//-----------------------------------------------------------------------------------------------------
//																
//									 	Tkmatik sp z o.o.
//
//	Name					:		FB_Load
//	Author					:		AM
//	Release Date			:		12.01.2022
//	Current ver				:		v 0.1
// 	Last correction 		:		12.01.2022
// 
//	Description				:
//		Special FB for loading structures from BINARY files						
//
//	Requared hardware		:
//
// 	Configuration			:
//
//
//-----------------------------------------------------------------------------------------------------

FUNCTION_BLOCK FB_Load
VAR_INPUT
	sFilePath											:	STRING(255);					//	File path (e.g. 'C:\1.txt')
	pStructAdr											:	PVOID;                          //	Pointer on data struct
	udiStructSize										:	UDINT;                          //	Size of datastruct
	bExecute											:	BOOL;                           //
END_VAR                                                                                     
VAR_OUTPUT                                                                                  
	bBusy												:	BOOL;                           //	FB is Busy
	bDone												:	BOOL;                           //	Load cycle done, DATA actual 
	bError												:	BOOL;                           //	Flag error
	nErrId												:	UDINT;                          //	Error ID
END_VAR                                                                                     
VAR                                                                                         
	fbFileOpen											:	FB_FileOpen;                    //	FB for opening 
	fbFileClose											:	FB_FileClose;                   //	FB for closing
	fbFileRead											:	FB_FileRead;                    //	FB for reading
	hFile												:	UINT;                           //	File hendler
	eMainCase											:	E_FileOpSteps;                  //	Main cycle case value
	rtExecute											:	R_TRIG;                         //	Rtrig for start
END_VAR

ACT_FBs();
ACT_Main();

ACTION ACT_FBs:
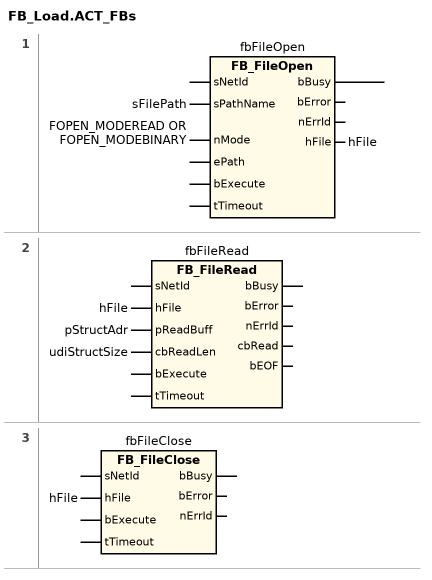
// NETWORK 1
fbFileOpen(sPathName := sFilePath, nMode := FOPEN_MODEREAD OR FOPEN_MODEBINARY, hFile => hFile); // FB_FileOpen

// NETWORK 2
fbFileRead(hFile := hFile, pReadBuff := pStructAdr, cbReadLen := udiStructSize); // FB_FileRead

// NETWORK 3
fbFileClose(hFile := hFile); // FB_FileClose
END_ACTION

ACTION ACT_Main:
rtExecute(CLK:=bExecute);
IF (NOT bExecute) THEN
	bDone												:=	FALSE;
END_IF

CASE eMainCase OF
	E_FileOpSteps.eNop:
		fbFileClose.bExecute							:=	FALSE;
		fbFileOpen.bExecute								:=	FALSE;
		fbFileRead.bExecute								:=	FALSE;
		bBusy											:=	FALSE;
		
		IF (rtExecute.Q) THEN
			bError										:=	FALSE;
			nErrId										:=	0;
			eMainCase									:=	E_FileOpSteps.eStartOpen;
			bBusy										:=	TRUE;
		END_IF
		
	E_FileOpSteps.eStartOpen:
		fbFileOpen.bExecute								:=	TRUE;
		eMainCase										:=	E_FileOpSteps.eWaitOpen;

	E_FileOpSteps.eWaitOpen:
		IF (fbFileOpen.bError) THEN
			bError										:=	TRUE;
			nErrId										:=	10;
			eMainCase									:=	E_FileOpSteps.eNop;
		ELSIF (NOT fbFileOpen.bBusy) THEN
			fbFileOpen.bExecute							:=	FALSE;
			eMainCase									:=	E_FileOpSteps.eStartOper;
		END_IF
		
	E_FileOpSteps.eStartOper:
		fbFileRead.bExecute								:=	TRUE;
		eMainCase										:=	E_FileOpSteps.eWaitOper;
		
	E_FileOpSteps.eWaitOper:
		IF (fbFileRead.bError) THEN
			bError										:=	TRUE;
			nErrId										:=	20;
			eMainCase									:=	E_FileOpSteps.eNop;
		ELSIF (NOT fbFileRead.bBusy) THEN
			fbFileRead.bExecute							:=	FALSE;
			eMainCase									:=	E_FileOpSteps.eStartClose;
		END_IF
		
	E_FileOpSteps.eStartClose:
		fbFileClose.bExecute							:=	TRUE;
		eMainCase										:=	E_FileOpSteps.eWaitClose;
	
	E_FileOpSteps.eWaitClose:
		IF (fbFileClose.bError) THEN
			bError										:=	TRUE;
			nErrId										:=	30;
			eMainCase									:=	E_FileOpSteps.eNop;
		ELSIF (NOT fbFileClose.bBusy) THEN
			fbFileClose.bExecute						:=	FALSE;
			bDone										:=	TRUE;
			eMainCase									:=	E_FileOpSteps.eNop;
		END_IF	
		
END_CASE
END_ACTION

END_FUNCTION_BLOCK

(* stored: Version 1.1.0.1, ProductVersion 3.1.4026.13, FileIdentifier 5faf5f79573d9a67dcb9c8edb448f1cb81efddc9, FileSignature 897c566a3b8ef87bced77a513133b1a500c63ef21e96527a5ed22cdf2df8e1183faace0e94b4b6bf971988f7875f5647288c4fcd91cd29e7fb1449694dde581b1331ddb47ae76f6ebd2577d4b020d96dfcc67e63d471be6cc7347f65c722611b793755998cedd9d76f72e2c1d1322230e85e8bf1dd43620df23319f0f6111f8651c849c01483dfe9d50b1d633ceb53c04cb56db5c7aac4461c4e32afafa695a1a63b645c24b715a8b2661a5cd8cb768623f99edf155c15e67da9b10d22c670361a7950ca5f428089c9c9c7d96b87b6a6110e80a544c11098adc96aff225fa7cb9c0fd4e90d5fdd6346cfbacf16d29becd85455e4e147ca932a3a1cd33d81fd02
   POU FB_Load: Id {809a43ef-8203-42f3-a062-b9c9cb97d64f}, SpecialFunc None
   Action ACT_FBs: Id {4ec5fe04-ef98-45ea-aeb1-905b3e8aec14}
   Action ACT_Main: Id {fc127786-59ff-4b69-a534-8476263b3645} *)
